// ============================================
// DB_RecipeProgram9 - Checksum Test
// Lines: 254
// CHUNKS: 10 x 100
// Generated by SpinningCam  [2026-08-14 11:34:49]
// ============================================
//
// --- MAKINE AYARLARI ---
// Machine Origin  : X=0.0, Z=0.0
// Axis Direction  : X=NORMAL, Z=NORMAL
// Output Mode     : RADIUS
// G54 Offset      : X=0.0, Z=0.0
// Home            : X=300.0, Z=150.0
// Retract         : X=50.0, Z=50.0
//
// --- PARCA / BLANK ---
// Blank Radius    : 0.0 mm
// Blank Z Shift   : 0.0 mm
// Final Thickness : 2.0 mm
// Min Safety Gap  : 0.0 mm
//
// --- MANDREL POZISYON ---
// Mandrel Offset  : X=0.0, Z=0.0
// Mandrel Rot     : Rx=0.0, Ry=0.0, Rz=0.0
// ============================================

DATA_BLOCK "DB_RecipeProgram9"
{ S7_Optimized_Access := 'FALSE' }
VERSION : 0.2
UNLINKED
NON_RETAIN
    VAR
        Header : "RecipeHeader";
        Lines1  : Array[0..99] of "RecipeLine";  // global lines 0..99
        Lines2  : Array[0..99] of "RecipeLine";  // global lines 100..199
        Lines3  : Array[0..99] of "RecipeLine";  // global lines 200..299
        Lines4  : Array[0..99] of "RecipeLine";  // global lines 300..399
        Lines5  : Array[0..99] of "RecipeLine";  // global lines 400..499
        Lines6  : Array[0..99] of "RecipeLine";  // global lines 500..599
        Lines7  : Array[0..99] of "RecipeLine";  // global lines 600..699
        Lines8  : Array[0..99] of "RecipeLine";  // global lines 700..799
        Lines9  : Array[0..99] of "RecipeLine";  // global lines 800..899
        Lines10 : Array[0..99] of "RecipeLine";  // global lines 900..999
    END_VAR
BEGIN
    // Header
    Header.sName := 'Checksum Test';
    Header.LineCount := 254;
    Header.Valid := TRUE;
    Header.PreScanned := FALSE;
    Header.MinX := 10.000;
    Header.MaxX := 134.500;
    Header.MinZ := 10.200;
    Header.MaxZ := 60.000;

    // --- Tool table (CAM-authored) ---
    Header.ProvidesToolConfig := TRUE;
    Header.ToolCount := 1;
    Header.AutoCalcAngles := TRUE;
    Header.ToolCode_List[1] := 101;
    Header.ToolCode_List[2] := 0;  // unused
    Header.ToolCode_List[3] := 0;  // unused
    Header.ToolCode_List[4] := 0;  // unused
    Header.ToolAngle_List[1] := 0.0;
    Header.ToolAngle_List[2] := 0.0;
    Header.ToolAngle_List[3] := 0.0;
    Header.ToolAngle_List[4] := 0.0;

    // --- Integrity ---
    // Order-sensitive sum over CMD+Param+F of lines 0..LineCount-1.
    // The PLC recomputes it after reassembling the chunks and refuses
    // to run on a mismatch (16#0316). X/Z are excluded on purpose:
    // float32-vs-float64 rounding would eventually cry wolf.
    Header.ProvidesChecksum := TRUE;
    Header.Checksum := 9593624;

    // Recipe Lines (254 total)

    // --- Lines1 (global lines 0..99) ---
    Lines1[0].X := 0.000; Lines1[0].Z := 0.000; Lines1[0].F := 0; Lines1[0].CMD := 20; Lines1[0].Param := 100; // Spindle ON 1000 RPM
    Lines1[1].X := 0.000; Lines1[1].Z := 0.000; Lines1[1].F := 0; Lines1[1].CMD := 10; Lines1[1].Param := 101; // Tool Change T101
    Lines1[2].X := 10.000; Lines1[2].Z := 60.000; Lines1[2].F := 300; Lines1[2].CMD := 1; Lines1[2].Param := 0; // G1 Linear
    Lines1[3].X := 10.500; Lines1[3].Z := 59.800; Lines1[3].F := 300; Lines1[3].CMD := 1; Lines1[3].Param := 0; // G1 Linear
    Lines1[4].X := 11.000; Lines1[4].Z := 59.600; Lines1[4].F := 300; Lines1[4].CMD := 1; Lines1[4].Param := 0; // G1 Linear
    Lines1[5].X := 11.500; Lines1[5].Z := 59.400; Lines1[5].F := 300; Lines1[5].CMD := 1; Lines1[5].Param := 0; // G1 Linear
    Lines1[6].X := 12.000; Lines1[6].Z := 59.200; Lines1[6].F := 300; Lines1[6].CMD := 1; Lines1[6].Param := 0; // G1 Linear
    Lines1[7].X := 12.500; Lines1[7].Z := 59.000; Lines1[7].F := 300; Lines1[7].CMD := 1; Lines1[7].Param := 0; // G1 Linear
    Lines1[8].X := 13.000; Lines1[8].Z := 58.800; Lines1[8].F := 300; Lines1[8].CMD := 1; Lines1[8].Param := 0; // G1 Linear
    Lines1[9].X := 13.500; Lines1[9].Z := 58.600; Lines1[9].F := 300; Lines1[9].CMD := 1; Lines1[9].Param := 0; // G1 Linear
    Lines1[10].X := 14.000; Lines1[10].Z := 58.400; Lines1[10].F := 300; Lines1[10].CMD := 1; Lines1[10].Param := 0; // G1 Linear
    Lines1[11].X := 14.500; Lines1[11].Z := 58.200; Lines1[11].F := 300; Lines1[11].CMD := 1; Lines1[11].Param := 0; // G1 Linear
    Lines1[12].X := 15.000; Lines1[12].Z := 58.000; Lines1[12].F := 300; Lines1[12].CMD := 1; Lines1[12].Param := 0; // G1 Linear
    Lines1[13].X := 15.500; Lines1[13].Z := 57.800; Lines1[13].F := 300; Lines1[13].CMD := 1; Lines1[13].Param := 0; // G1 Linear
    Lines1[14].X := 16.000; Lines1[14].Z := 57.600; Lines1[14].F := 300; Lines1[14].CMD := 1; Lines1[14].Param := 0; // G1 Linear
    Lines1[15].X := 16.500; Lines1[15].Z := 57.400; Lines1[15].F := 300; Lines1[15].CMD := 1; Lines1[15].Param := 0; // G1 Linear
    Lines1[16].X := 17.000; Lines1[16].Z := 57.200; Lines1[16].F := 300; Lines1[16].CMD := 1; Lines1[16].Param := 0; // G1 Linear
    Lines1[17].X := 17.500; Lines1[17].Z := 57.000; Lines1[17].F := 300; Lines1[17].CMD := 1; Lines1[17].Param := 0; // G1 Linear
    Lines1[18].X := 18.000; Lines1[18].Z := 56.800; Lines1[18].F := 300; Lines1[18].CMD := 1; Lines1[18].Param := 0; // G1 Linear
    Lines1[19].X := 18.500; Lines1[19].Z := 56.600; Lines1[19].F := 300; Lines1[19].CMD := 1; Lines1[19].Param := 0; // G1 Linear
    Lines1[20].X := 19.000; Lines1[20].Z := 56.400; Lines1[20].F := 300; Lines1[20].CMD := 1; Lines1[20].Param := 0; // G1 Linear
    Lines1[21].X := 19.500; Lines1[21].Z := 56.200; Lines1[21].F := 300; Lines1[21].CMD := 1; Lines1[21].Param := 0; // G1 Linear
    Lines1[22].X := 20.000; Lines1[22].Z := 56.000; Lines1[22].F := 300; Lines1[22].CMD := 1; Lines1[22].Param := 0; // G1 Linear
    Lines1[23].X := 20.500; Lines1[23].Z := 55.800; Lines1[23].F := 300; Lines1[23].CMD := 1; Lines1[23].Param := 0; // G1 Linear
    Lines1[24].X := 21.000; Lines1[24].Z := 55.600; Lines1[24].F := 300; Lines1[24].CMD := 1; Lines1[24].Param := 0; // G1 Linear
    Lines1[25].X := 21.500; Lines1[25].Z := 55.400; Lines1[25].F := 300; Lines1[25].CMD := 1; Lines1[25].Param := 0; // G1 Linear
    Lines1[26].X := 22.000; Lines1[26].Z := 55.200; Lines1[26].F := 300; Lines1[26].CMD := 1; Lines1[26].Param := 0; // G1 Linear
    Lines1[27].X := 22.500; Lines1[27].Z := 55.000; Lines1[27].F := 300; Lines1[27].CMD := 1; Lines1[27].Param := 0; // G1 Linear
    Lines1[28].X := 23.000; Lines1[28].Z := 54.800; Lines1[28].F := 300; Lines1[28].CMD := 1; Lines1[28].Param := 0; // G1 Linear
    Lines1[29].X := 23.500; Lines1[29].Z := 54.600; Lines1[29].F := 300; Lines1[29].CMD := 1; Lines1[29].Param := 0; // G1 Linear
    Lines1[30].X := 24.000; Lines1[30].Z := 54.400; Lines1[30].F := 300; Lines1[30].CMD := 1; Lines1[30].Param := 0; // G1 Linear
    Lines1[31].X := 24.500; Lines1[31].Z := 54.200; Lines1[31].F := 300; Lines1[31].CMD := 1; Lines1[31].Param := 0; // G1 Linear
    Lines1[32].X := 25.000; Lines1[32].Z := 54.000; Lines1[32].F := 300; Lines1[32].CMD := 1; Lines1[32].Param := 0; // G1 Linear
    Lines1[33].X := 25.500; Lines1[33].Z := 53.800; Lines1[33].F := 300; Lines1[33].CMD := 1; Lines1[33].Param := 0; // G1 Linear
    Lines1[34].X := 26.000; Lines1[34].Z := 53.600; Lines1[34].F := 300; Lines1[34].CMD := 1; Lines1[34].Param := 0; // G1 Linear
    Lines1[35].X := 26.500; Lines1[35].Z := 53.400; Lines1[35].F := 300; Lines1[35].CMD := 1; Lines1[35].Param := 0; // G1 Linear
    Lines1[36].X := 27.000; Lines1[36].Z := 53.200; Lines1[36].F := 300; Lines1[36].CMD := 1; Lines1[36].Param := 0; // G1 Linear
    Lines1[37].X := 27.500; Lines1[37].Z := 53.000; Lines1[37].F := 300; Lines1[37].CMD := 1; Lines1[37].Param := 0; // G1 Linear
    Lines1[38].X := 28.000; Lines1[38].Z := 52.800; Lines1[38].F := 300; Lines1[38].CMD := 1; Lines1[38].Param := 0; // G1 Linear
    Lines1[39].X := 28.500; Lines1[39].Z := 52.600; Lines1[39].F := 300; Lines1[39].CMD := 1; Lines1[39].Param := 0; // G1 Linear
    Lines1[40].X := 29.000; Lines1[40].Z := 52.400; Lines1[40].F := 300; Lines1[40].CMD := 1; Lines1[40].Param := 0; // G1 Linear
    Lines1[41].X := 29.500; Lines1[41].Z := 52.200; Lines1[41].F := 300; Lines1[41].CMD := 1; Lines1[41].Param := 0; // G1 Linear
    Lines1[42].X := 30.000; Lines1[42].Z := 52.000; Lines1[42].F := 300; Lines1[42].CMD := 1; Lines1[42].Param := 0; // G1 Linear
    Lines1[43].X := 30.500; Lines1[43].Z := 51.800; Lines1[43].F := 300; Lines1[43].CMD := 1; Lines1[43].Param := 0; // G1 Linear
    Lines1[44].X := 31.000; Lines1[44].Z := 51.600; Lines1[44].F := 300; Lines1[44].CMD := 1; Lines1[44].Param := 0; // G1 Linear
    Lines1[45].X := 31.500; Lines1[45].Z := 51.400; Lines1[45].F := 300; Lines1[45].CMD := 1; Lines1[45].Param := 0; // G1 Linear
    Lines1[46].X := 32.000; Lines1[46].Z := 51.200; Lines1[46].F := 300; Lines1[46].CMD := 1; Lines1[46].Param := 0; // G1 Linear
    Lines1[47].X := 32.500; Lines1[47].Z := 51.000; Lines1[47].F := 300; Lines1[47].CMD := 1; Lines1[47].Param := 0; // G1 Linear
    Lines1[48].X := 33.000; Lines1[48].Z := 50.800; Lines1[48].F := 300; Lines1[48].CMD := 1; Lines1[48].Param := 0; // G1 Linear
    Lines1[49].X := 33.500; Lines1[49].Z := 50.600; Lines1[49].F := 300; Lines1[49].CMD := 1; Lines1[49].Param := 0; // G1 Linear
    Lines1[50].X := 34.000; Lines1[50].Z := 50.400; Lines1[50].F := 300; Lines1[50].CMD := 1; Lines1[50].Param := 0; // G1 Linear
    Lines1[51].X := 34.500; Lines1[51].Z := 50.200; Lines1[51].F := 300; Lines1[51].CMD := 1; Lines1[51].Param := 0; // G1 Linear
    Lines1[52].X := 35.000; Lines1[52].Z := 50.000; Lines1[52].F := 300; Lines1[52].CMD := 1; Lines1[52].Param := 0; // G1 Linear
    Lines1[53].X := 35.500; Lines1[53].Z := 49.800; Lines1[53].F := 300; Lines1[53].CMD := 1; Lines1[53].Param := 0; // G1 Linear
    Lines1[54].X := 36.000; Lines1[54].Z := 49.600; Lines1[54].F := 300; Lines1[54].CMD := 1; Lines1[54].Param := 0; // G1 Linear
    Lines1[55].X := 36.500; Lines1[55].Z := 49.400; Lines1[55].F := 300; Lines1[55].CMD := 1; Lines1[55].Param := 0; // G1 Linear
    Lines1[56].X := 37.000; Lines1[56].Z := 49.200; Lines1[56].F := 300; Lines1[56].CMD := 1; Lines1[56].Param := 0; // G1 Linear
    Lines1[57].X := 37.500; Lines1[57].Z := 49.000; Lines1[57].F := 300; Lines1[57].CMD := 1; Lines1[57].Param := 0; // G1 Linear
    Lines1[58].X := 38.000; Lines1[58].Z := 48.800; Lines1[58].F := 300; Lines1[58].CMD := 1; Lines1[58].Param := 0; // G1 Linear
    Lines1[59].X := 38.500; Lines1[59].Z := 48.600; Lines1[59].F := 300; Lines1[59].CMD := 1; Lines1[59].Param := 0; // G1 Linear
    Lines1[60].X := 39.000; Lines1[60].Z := 48.400; Lines1[60].F := 300; Lines1[60].CMD := 1; Lines1[60].Param := 0; // G1 Linear
    Lines1[61].X := 39.500; Lines1[61].Z := 48.200; Lines1[61].F := 300; Lines1[61].CMD := 1; Lines1[61].Param := 0; // G1 Linear
    Lines1[62].X := 40.000; Lines1[62].Z := 48.000; Lines1[62].F := 300; Lines1[62].CMD := 1; Lines1[62].Param := 0; // G1 Linear
    Lines1[63].X := 40.500; Lines1[63].Z := 47.800; Lines1[63].F := 300; Lines1[63].CMD := 1; Lines1[63].Param := 0; // G1 Linear
    Lines1[64].X := 41.000; Lines1[64].Z := 47.600; Lines1[64].F := 300; Lines1[64].CMD := 1; Lines1[64].Param := 0; // G1 Linear
    Lines1[65].X := 41.500; Lines1[65].Z := 47.400; Lines1[65].F := 300; Lines1[65].CMD := 1; Lines1[65].Param := 0; // G1 Linear
    Lines1[66].X := 42.000; Lines1[66].Z := 47.200; Lines1[66].F := 300; Lines1[66].CMD := 1; Lines1[66].Param := 0; // G1 Linear
    Lines1[67].X := 42.500; Lines1[67].Z := 47.000; Lines1[67].F := 300; Lines1[67].CMD := 1; Lines1[67].Param := 0; // G1 Linear
    Lines1[68].X := 43.000; Lines1[68].Z := 46.800; Lines1[68].F := 300; Lines1[68].CMD := 1; Lines1[68].Param := 0; // G1 Linear
    Lines1[69].X := 43.500; Lines1[69].Z := 46.600; Lines1[69].F := 300; Lines1[69].CMD := 1; Lines1[69].Param := 0; // G1 Linear
    Lines1[70].X := 44.000; Lines1[70].Z := 46.400; Lines1[70].F := 300; Lines1[70].CMD := 1; Lines1[70].Param := 0; // G1 Linear
    Lines1[71].X := 44.500; Lines1[71].Z := 46.200; Lines1[71].F := 300; Lines1[71].CMD := 1; Lines1[71].Param := 0; // G1 Linear
    Lines1[72].X := 45.000; Lines1[72].Z := 46.000; Lines1[72].F := 300; Lines1[72].CMD := 1; Lines1[72].Param := 0; // G1 Linear
    Lines1[73].X := 45.500; Lines1[73].Z := 45.800; Lines1[73].F := 300; Lines1[73].CMD := 1; Lines1[73].Param := 0; // G1 Linear
    Lines1[74].X := 46.000; Lines1[74].Z := 45.600; Lines1[74].F := 300; Lines1[74].CMD := 1; Lines1[74].Param := 0; // G1 Linear
    Lines1[75].X := 46.500; Lines1[75].Z := 45.400; Lines1[75].F := 300; Lines1[75].CMD := 1; Lines1[75].Param := 0; // G1 Linear
    Lines1[76].X := 47.000; Lines1[76].Z := 45.200; Lines1[76].F := 300; Lines1[76].CMD := 1; Lines1[76].Param := 0; // G1 Linear
    Lines1[77].X := 47.500; Lines1[77].Z := 45.000; Lines1[77].F := 300; Lines1[77].CMD := 1; Lines1[77].Param := 0; // G1 Linear
    Lines1[78].X := 48.000; Lines1[78].Z := 44.800; Lines1[78].F := 300; Lines1[78].CMD := 1; Lines1[78].Param := 0; // G1 Linear
    Lines1[79].X := 48.500; Lines1[79].Z := 44.600; Lines1[79].F := 300; Lines1[79].CMD := 1; Lines1[79].Param := 0; // G1 Linear
    Lines1[80].X := 49.000; Lines1[80].Z := 44.400; Lines1[80].F := 300; Lines1[80].CMD := 1; Lines1[80].Param := 0; // G1 Linear
    Lines1[81].X := 49.500; Lines1[81].Z := 44.200; Lines1[81].F := 300; Lines1[81].CMD := 1; Lines1[81].Param := 0; // G1 Linear
    Lines1[82].X := 50.000; Lines1[82].Z := 44.000; Lines1[82].F := 300; Lines1[82].CMD := 1; Lines1[82].Param := 0; // G1 Linear
    Lines1[83].X := 50.500; Lines1[83].Z := 43.800; Lines1[83].F := 300; Lines1[83].CMD := 1; Lines1[83].Param := 0; // G1 Linear
    Lines1[84].X := 51.000; Lines1[84].Z := 43.600; Lines1[84].F := 300; Lines1[84].CMD := 1; Lines1[84].Param := 0; // G1 Linear
    Lines1[85].X := 51.500; Lines1[85].Z := 43.400; Lines1[85].F := 300; Lines1[85].CMD := 1; Lines1[85].Param := 0; // G1 Linear
    Lines1[86].X := 52.000; Lines1[86].Z := 43.200; Lines1[86].F := 300; Lines1[86].CMD := 1; Lines1[86].Param := 0; // G1 Linear
    Lines1[87].X := 52.500; Lines1[87].Z := 43.000; Lines1[87].F := 300; Lines1[87].CMD := 1; Lines1[87].Param := 0; // G1 Linear
    Lines1[88].X := 53.000; Lines1[88].Z := 42.800; Lines1[88].F := 300; Lines1[88].CMD := 1; Lines1[88].Param := 0; // G1 Linear
    Lines1[89].X := 53.500; Lines1[89].Z := 42.600; Lines1[89].F := 300; Lines1[89].CMD := 1; Lines1[89].Param := 0; // G1 Linear
    Lines1[90].X := 54.000; Lines1[90].Z := 42.400; Lines1[90].F := 300; Lines1[90].CMD := 1; Lines1[90].Param := 0; // G1 Linear
    Lines1[91].X := 54.500; Lines1[91].Z := 42.200; Lines1[91].F := 300; Lines1[91].CMD := 1; Lines1[91].Param := 0; // G1 Linear
    Lines1[92].X := 55.000; Lines1[92].Z := 42.000; Lines1[92].F := 300; Lines1[92].CMD := 1; Lines1[92].Param := 0; // G1 Linear
    Lines1[93].X := 55.500; Lines1[93].Z := 41.800; Lines1[93].F := 300; Lines1[93].CMD := 1; Lines1[93].Param := 0; // G1 Linear
    Lines1[94].X := 56.000; Lines1[94].Z := 41.600; Lines1[94].F := 300; Lines1[94].CMD := 1; Lines1[94].Param := 0; // G1 Linear
    Lines1[95].X := 56.500; Lines1[95].Z := 41.400; Lines1[95].F := 300; Lines1[95].CMD := 1; Lines1[95].Param := 0; // G1 Linear
    Lines1[96].X := 57.000; Lines1[96].Z := 41.200; Lines1[96].F := 300; Lines1[96].CMD := 1; Lines1[96].Param := 0; // G1 Linear
    Lines1[97].X := 57.500; Lines1[97].Z := 41.000; Lines1[97].F := 300; Lines1[97].CMD := 1; Lines1[97].Param := 0; // G1 Linear
    Lines1[98].X := 58.000; Lines1[98].Z := 40.800; Lines1[98].F := 300; Lines1[98].CMD := 1; Lines1[98].Param := 0; // G1 Linear
    Lines1[99].X := 58.500; Lines1[99].Z := 40.600; Lines1[99].F := 300; Lines1[99].CMD := 1; Lines1[99].Param := 0; // G1 Linear

    // --- Lines2 (global lines 100..199) ---
    Lines2[0].X := 59.000; Lines2[0].Z := 40.400; Lines2[0].F := 300; Lines2[0].CMD := 1; Lines2[0].Param := 0; // G1 Linear
    Lines2[1].X := 59.500; Lines2[1].Z := 40.200; Lines2[1].F := 300; Lines2[1].CMD := 1; Lines2[1].Param := 0; // G1 Linear
    Lines2[2].X := 60.000; Lines2[2].Z := 40.000; Lines2[2].F := 300; Lines2[2].CMD := 1; Lines2[2].Param := 0; // G1 Linear
    Lines2[3].X := 60.500; Lines2[3].Z := 39.800; Lines2[3].F := 300; Lines2[3].CMD := 1; Lines2[3].Param := 0; // G1 Linear
    Lines2[4].X := 61.000; Lines2[4].Z := 39.600; Lines2[4].F := 300; Lines2[4].CMD := 1; Lines2[4].Param := 0; // G1 Linear
    Lines2[5].X := 61.500; Lines2[5].Z := 39.400; Lines2[5].F := 300; Lines2[5].CMD := 1; Lines2[5].Param := 0; // G1 Linear
    Lines2[6].X := 62.000; Lines2[6].Z := 39.200; Lines2[6].F := 300; Lines2[6].CMD := 1; Lines2[6].Param := 0; // G1 Linear
    Lines2[7].X := 62.500; Lines2[7].Z := 39.000; Lines2[7].F := 300; Lines2[7].CMD := 1; Lines2[7].Param := 0; // G1 Linear
    Lines2[8].X := 63.000; Lines2[8].Z := 38.800; Lines2[8].F := 300; Lines2[8].CMD := 1; Lines2[8].Param := 0; // G1 Linear
    Lines2[9].X := 63.500; Lines2[9].Z := 38.600; Lines2[9].F := 300; Lines2[9].CMD := 1; Lines2[9].Param := 0; // G1 Linear
    Lines2[10].X := 64.000; Lines2[10].Z := 38.400; Lines2[10].F := 300; Lines2[10].CMD := 1; Lines2[10].Param := 0; // G1 Linear
    Lines2[11].X := 64.500; Lines2[11].Z := 38.200; Lines2[11].F := 300; Lines2[11].CMD := 1; Lines2[11].Param := 0; // G1 Linear
    Lines2[12].X := 65.000; Lines2[12].Z := 38.000; Lines2[12].F := 300; Lines2[12].CMD := 1; Lines2[12].Param := 0; // G1 Linear
    Lines2[13].X := 65.500; Lines2[13].Z := 37.800; Lines2[13].F := 300; Lines2[13].CMD := 1; Lines2[13].Param := 0; // G1 Linear
    Lines2[14].X := 66.000; Lines2[14].Z := 37.600; Lines2[14].F := 300; Lines2[14].CMD := 1; Lines2[14].Param := 0; // G1 Linear
    Lines2[15].X := 66.500; Lines2[15].Z := 37.400; Lines2[15].F := 300; Lines2[15].CMD := 1; Lines2[15].Param := 0; // G1 Linear
    Lines2[16].X := 67.000; Lines2[16].Z := 37.200; Lines2[16].F := 300; Lines2[16].CMD := 1; Lines2[16].Param := 0; // G1 Linear
    Lines2[17].X := 67.500; Lines2[17].Z := 37.000; Lines2[17].F := 300; Lines2[17].CMD := 1; Lines2[17].Param := 0; // G1 Linear
    Lines2[18].X := 68.000; Lines2[18].Z := 36.800; Lines2[18].F := 300; Lines2[18].CMD := 1; Lines2[18].Param := 0; // G1 Linear
    Lines2[19].X := 68.500; Lines2[19].Z := 36.600; Lines2[19].F := 300; Lines2[19].CMD := 1; Lines2[19].Param := 0; // G1 Linear
    Lines2[20].X := 69.000; Lines2[20].Z := 36.400; Lines2[20].F := 300; Lines2[20].CMD := 1; Lines2[20].Param := 0; // G1 Linear
    Lines2[21].X := 69.500; Lines2[21].Z := 36.200; Lines2[21].F := 300; Lines2[21].CMD := 1; Lines2[21].Param := 0; // G1 Linear
    Lines2[22].X := 70.000; Lines2[22].Z := 36.000; Lines2[22].F := 300; Lines2[22].CMD := 1; Lines2[22].Param := 0; // G1 Linear
    Lines2[23].X := 70.500; Lines2[23].Z := 35.800; Lines2[23].F := 300; Lines2[23].CMD := 1; Lines2[23].Param := 0; // G1 Linear
    Lines2[24].X := 71.000; Lines2[24].Z := 35.600; Lines2[24].F := 300; Lines2[24].CMD := 1; Lines2[24].Param := 0; // G1 Linear
    Lines2[25].X := 71.500; Lines2[25].Z := 35.400; Lines2[25].F := 300; Lines2[25].CMD := 1; Lines2[25].Param := 0; // G1 Linear
    Lines2[26].X := 72.000; Lines2[26].Z := 35.200; Lines2[26].F := 300; Lines2[26].CMD := 1; Lines2[26].Param := 0; // G1 Linear
    Lines2[27].X := 72.500; Lines2[27].Z := 35.000; Lines2[27].F := 300; Lines2[27].CMD := 1; Lines2[27].Param := 0; // G1 Linear
    Lines2[28].X := 73.000; Lines2[28].Z := 34.800; Lines2[28].F := 300; Lines2[28].CMD := 1; Lines2[28].Param := 0; // G1 Linear
    Lines2[29].X := 73.500; Lines2[29].Z := 34.600; Lines2[29].F := 300; Lines2[29].CMD := 1; Lines2[29].Param := 0; // G1 Linear
    Lines2[30].X := 74.000; Lines2[30].Z := 34.400; Lines2[30].F := 300; Lines2[30].CMD := 1; Lines2[30].Param := 0; // G1 Linear
    Lines2[31].X := 74.500; Lines2[31].Z := 34.200; Lines2[31].F := 300; Lines2[31].CMD := 1; Lines2[31].Param := 0; // G1 Linear
    Lines2[32].X := 75.000; Lines2[32].Z := 34.000; Lines2[32].F := 300; Lines2[32].CMD := 1; Lines2[32].Param := 0; // G1 Linear
    Lines2[33].X := 75.500; Lines2[33].Z := 33.800; Lines2[33].F := 300; Lines2[33].CMD := 1; Lines2[33].Param := 0; // G1 Linear
    Lines2[34].X := 76.000; Lines2[34].Z := 33.600; Lines2[34].F := 300; Lines2[34].CMD := 1; Lines2[34].Param := 0; // G1 Linear
    Lines2[35].X := 76.500; Lines2[35].Z := 33.400; Lines2[35].F := 300; Lines2[35].CMD := 1; Lines2[35].Param := 0; // G1 Linear
    Lines2[36].X := 77.000; Lines2[36].Z := 33.200; Lines2[36].F := 300; Lines2[36].CMD := 1; Lines2[36].Param := 0; // G1 Linear
    Lines2[37].X := 77.500; Lines2[37].Z := 33.000; Lines2[37].F := 300; Lines2[37].CMD := 1; Lines2[37].Param := 0; // G1 Linear
    Lines2[38].X := 78.000; Lines2[38].Z := 32.800; Lines2[38].F := 300; Lines2[38].CMD := 1; Lines2[38].Param := 0; // G1 Linear
    Lines2[39].X := 78.500; Lines2[39].Z := 32.600; Lines2[39].F := 300; Lines2[39].CMD := 1; Lines2[39].Param := 0; // G1 Linear
    Lines2[40].X := 79.000; Lines2[40].Z := 32.400; Lines2[40].F := 300; Lines2[40].CMD := 1; Lines2[40].Param := 0; // G1 Linear
    Lines2[41].X := 79.500; Lines2[41].Z := 32.200; Lines2[41].F := 300; Lines2[41].CMD := 1; Lines2[41].Param := 0; // G1 Linear
    Lines2[42].X := 80.000; Lines2[42].Z := 32.000; Lines2[42].F := 300; Lines2[42].CMD := 1; Lines2[42].Param := 0; // G1 Linear
    Lines2[43].X := 80.500; Lines2[43].Z := 31.800; Lines2[43].F := 300; Lines2[43].CMD := 1; Lines2[43].Param := 0; // G1 Linear
    Lines2[44].X := 81.000; Lines2[44].Z := 31.600; Lines2[44].F := 300; Lines2[44].CMD := 1; Lines2[44].Param := 0; // G1 Linear
    Lines2[45].X := 81.500; Lines2[45].Z := 31.400; Lines2[45].F := 300; Lines2[45].CMD := 1; Lines2[45].Param := 0; // G1 Linear
    Lines2[46].X := 82.000; Lines2[46].Z := 31.200; Lines2[46].F := 300; Lines2[46].CMD := 1; Lines2[46].Param := 0; // G1 Linear
    Lines2[47].X := 82.500; Lines2[47].Z := 31.000; Lines2[47].F := 300; Lines2[47].CMD := 1; Lines2[47].Param := 0; // G1 Linear
    Lines2[48].X := 83.000; Lines2[48].Z := 30.800; Lines2[48].F := 300; Lines2[48].CMD := 1; Lines2[48].Param := 0; // G1 Linear
    Lines2[49].X := 83.500; Lines2[49].Z := 30.600; Lines2[49].F := 300; Lines2[49].CMD := 1; Lines2[49].Param := 0; // G1 Linear
    Lines2[50].X := 84.000; Lines2[50].Z := 30.400; Lines2[50].F := 300; Lines2[50].CMD := 1; Lines2[50].Param := 0; // G1 Linear
    Lines2[51].X := 84.500; Lines2[51].Z := 30.200; Lines2[51].F := 300; Lines2[51].CMD := 1; Lines2[51].Param := 0; // G1 Linear
    Lines2[52].X := 85.000; Lines2[52].Z := 30.000; Lines2[52].F := 300; Lines2[52].CMD := 1; Lines2[52].Param := 0; // G1 Linear
    Lines2[53].X := 85.500; Lines2[53].Z := 29.800; Lines2[53].F := 300; Lines2[53].CMD := 1; Lines2[53].Param := 0; // G1 Linear
    Lines2[54].X := 86.000; Lines2[54].Z := 29.600; Lines2[54].F := 300; Lines2[54].CMD := 1; Lines2[54].Param := 0; // G1 Linear
    Lines2[55].X := 86.500; Lines2[55].Z := 29.400; Lines2[55].F := 300; Lines2[55].CMD := 1; Lines2[55].Param := 0; // G1 Linear
    Lines2[56].X := 87.000; Lines2[56].Z := 29.200; Lines2[56].F := 300; Lines2[56].CMD := 1; Lines2[56].Param := 0; // G1 Linear
    Lines2[57].X := 87.500; Lines2[57].Z := 29.000; Lines2[57].F := 300; Lines2[57].CMD := 1; Lines2[57].Param := 0; // G1 Linear
    Lines2[58].X := 88.000; Lines2[58].Z := 28.800; Lines2[58].F := 300; Lines2[58].CMD := 1; Lines2[58].Param := 0; // G1 Linear
    Lines2[59].X := 88.500; Lines2[59].Z := 28.600; Lines2[59].F := 300; Lines2[59].CMD := 1; Lines2[59].Param := 0; // G1 Linear
    Lines2[60].X := 89.000; Lines2[60].Z := 28.400; Lines2[60].F := 300; Lines2[60].CMD := 1; Lines2[60].Param := 0; // G1 Linear
    Lines2[61].X := 89.500; Lines2[61].Z := 28.200; Lines2[61].F := 300; Lines2[61].CMD := 1; Lines2[61].Param := 0; // G1 Linear
    Lines2[62].X := 90.000; Lines2[62].Z := 28.000; Lines2[62].F := 300; Lines2[62].CMD := 1; Lines2[62].Param := 0; // G1 Linear
    Lines2[63].X := 90.500; Lines2[63].Z := 27.800; Lines2[63].F := 300; Lines2[63].CMD := 1; Lines2[63].Param := 0; // G1 Linear
    Lines2[64].X := 91.000; Lines2[64].Z := 27.600; Lines2[64].F := 300; Lines2[64].CMD := 1; Lines2[64].Param := 0; // G1 Linear
    Lines2[65].X := 91.500; Lines2[65].Z := 27.400; Lines2[65].F := 300; Lines2[65].CMD := 1; Lines2[65].Param := 0; // G1 Linear
    Lines2[66].X := 92.000; Lines2[66].Z := 27.200; Lines2[66].F := 300; Lines2[66].CMD := 1; Lines2[66].Param := 0; // G1 Linear
    Lines2[67].X := 92.500; Lines2[67].Z := 27.000; Lines2[67].F := 300; Lines2[67].CMD := 1; Lines2[67].Param := 0; // G1 Linear
    Lines2[68].X := 93.000; Lines2[68].Z := 26.800; Lines2[68].F := 300; Lines2[68].CMD := 1; Lines2[68].Param := 0; // G1 Linear
    Lines2[69].X := 93.500; Lines2[69].Z := 26.600; Lines2[69].F := 300; Lines2[69].CMD := 1; Lines2[69].Param := 0; // G1 Linear
    Lines2[70].X := 94.000; Lines2[70].Z := 26.400; Lines2[70].F := 300; Lines2[70].CMD := 1; Lines2[70].Param := 0; // G1 Linear
    Lines2[71].X := 94.500; Lines2[71].Z := 26.200; Lines2[71].F := 300; Lines2[71].CMD := 1; Lines2[71].Param := 0; // G1 Linear
    Lines2[72].X := 95.000; Lines2[72].Z := 26.000; Lines2[72].F := 300; Lines2[72].CMD := 1; Lines2[72].Param := 0; // G1 Linear
    Lines2[73].X := 95.500; Lines2[73].Z := 25.800; Lines2[73].F := 300; Lines2[73].CMD := 1; Lines2[73].Param := 0; // G1 Linear
    Lines2[74].X := 96.000; Lines2[74].Z := 25.600; Lines2[74].F := 300; Lines2[74].CMD := 1; Lines2[74].Param := 0; // G1 Linear
    Lines2[75].X := 96.500; Lines2[75].Z := 25.400; Lines2[75].F := 300; Lines2[75].CMD := 1; Lines2[75].Param := 0; // G1 Linear
    Lines2[76].X := 97.000; Lines2[76].Z := 25.200; Lines2[76].F := 300; Lines2[76].CMD := 1; Lines2[76].Param := 0; // G1 Linear
    Lines2[77].X := 97.500; Lines2[77].Z := 25.000; Lines2[77].F := 300; Lines2[77].CMD := 1; Lines2[77].Param := 0; // G1 Linear
    Lines2[78].X := 98.000; Lines2[78].Z := 24.800; Lines2[78].F := 300; Lines2[78].CMD := 1; Lines2[78].Param := 0; // G1 Linear
    Lines2[79].X := 98.500; Lines2[79].Z := 24.600; Lines2[79].F := 300; Lines2[79].CMD := 1; Lines2[79].Param := 0; // G1 Linear
    Lines2[80].X := 99.000; Lines2[80].Z := 24.400; Lines2[80].F := 300; Lines2[80].CMD := 1; Lines2[80].Param := 0; // G1 Linear
    Lines2[81].X := 99.500; Lines2[81].Z := 24.200; Lines2[81].F := 300; Lines2[81].CMD := 1; Lines2[81].Param := 0; // G1 Linear
    Lines2[82].X := 100.000; Lines2[82].Z := 24.000; Lines2[82].F := 300; Lines2[82].CMD := 1; Lines2[82].Param := 0; // G1 Linear
    Lines2[83].X := 100.500; Lines2[83].Z := 23.800; Lines2[83].F := 300; Lines2[83].CMD := 1; Lines2[83].Param := 0; // G1 Linear
    Lines2[84].X := 101.000; Lines2[84].Z := 23.600; Lines2[84].F := 300; Lines2[84].CMD := 1; Lines2[84].Param := 0; // G1 Linear
    Lines2[85].X := 101.500; Lines2[85].Z := 23.400; Lines2[85].F := 300; Lines2[85].CMD := 1; Lines2[85].Param := 0; // G1 Linear
    Lines2[86].X := 102.000; Lines2[86].Z := 23.200; Lines2[86].F := 300; Lines2[86].CMD := 1; Lines2[86].Param := 0; // G1 Linear
    Lines2[87].X := 102.500; Lines2[87].Z := 23.000; Lines2[87].F := 300; Lines2[87].CMD := 1; Lines2[87].Param := 0; // G1 Linear
    Lines2[88].X := 103.000; Lines2[88].Z := 22.800; Lines2[88].F := 300; Lines2[88].CMD := 1; Lines2[88].Param := 0; // G1 Linear
    Lines2[89].X := 103.500; Lines2[89].Z := 22.600; Lines2[89].F := 300; Lines2[89].CMD := 1; Lines2[89].Param := 0; // G1 Linear
    Lines2[90].X := 104.000; Lines2[90].Z := 22.400; Lines2[90].F := 300; Lines2[90].CMD := 1; Lines2[90].Param := 0; // G1 Linear
    Lines2[91].X := 104.500; Lines2[91].Z := 22.200; Lines2[91].F := 300; Lines2[91].CMD := 1; Lines2[91].Param := 0; // G1 Linear
    Lines2[92].X := 105.000; Lines2[92].Z := 22.000; Lines2[92].F := 300; Lines2[92].CMD := 1; Lines2[92].Param := 0; // G1 Linear
    Lines2[93].X := 105.500; Lines2[93].Z := 21.800; Lines2[93].F := 300; Lines2[93].CMD := 1; Lines2[93].Param := 0; // G1 Linear
    Lines2[94].X := 106.000; Lines2[94].Z := 21.600; Lines2[94].F := 300; Lines2[94].CMD := 1; Lines2[94].Param := 0; // G1 Linear
    Lines2[95].X := 106.500; Lines2[95].Z := 21.400; Lines2[95].F := 300; Lines2[95].CMD := 1; Lines2[95].Param := 0; // G1 Linear
    Lines2[96].X := 107.000; Lines2[96].Z := 21.200; Lines2[96].F := 300; Lines2[96].CMD := 1; Lines2[96].Param := 0; // G1 Linear
    Lines2[97].X := 107.500; Lines2[97].Z := 21.000; Lines2[97].F := 300; Lines2[97].CMD := 1; Lines2[97].Param := 0; // G1 Linear
    Lines2[98].X := 108.000; Lines2[98].Z := 20.800; Lines2[98].F := 300; Lines2[98].CMD := 1; Lines2[98].Param := 0; // G1 Linear
    Lines2[99].X := 108.500; Lines2[99].Z := 20.600; Lines2[99].F := 300; Lines2[99].CMD := 1; Lines2[99].Param := 0; // G1 Linear

    // --- Lines3 (global lines 200..253) ---
    Lines3[0].X := 109.000; Lines3[0].Z := 20.400; Lines3[0].F := 300; Lines3[0].CMD := 1; Lines3[0].Param := 0; // G1 Linear
    Lines3[1].X := 109.500; Lines3[1].Z := 20.200; Lines3[1].F := 300; Lines3[1].CMD := 1; Lines3[1].Param := 0; // G1 Linear
    Lines3[2].X := 110.000; Lines3[2].Z := 20.000; Lines3[2].F := 300; Lines3[2].CMD := 1; Lines3[2].Param := 0; // G1 Linear
    Lines3[3].X := 110.500; Lines3[3].Z := 19.800; Lines3[3].F := 300; Lines3[3].CMD := 1; Lines3[3].Param := 0; // G1 Linear
    Lines3[4].X := 111.000; Lines3[4].Z := 19.600; Lines3[4].F := 300; Lines3[4].CMD := 1; Lines3[4].Param := 0; // G1 Linear
    Lines3[5].X := 111.500; Lines3[5].Z := 19.400; Lines3[5].F := 300; Lines3[5].CMD := 1; Lines3[5].Param := 0; // G1 Linear
    Lines3[6].X := 112.000; Lines3[6].Z := 19.200; Lines3[6].F := 300; Lines3[6].CMD := 1; Lines3[6].Param := 0; // G1 Linear
    Lines3[7].X := 112.500; Lines3[7].Z := 19.000; Lines3[7].F := 300; Lines3[7].CMD := 1; Lines3[7].Param := 0; // G1 Linear
    Lines3[8].X := 113.000; Lines3[8].Z := 18.800; Lines3[8].F := 300; Lines3[8].CMD := 1; Lines3[8].Param := 0; // G1 Linear
    Lines3[9].X := 113.500; Lines3[9].Z := 18.600; Lines3[9].F := 300; Lines3[9].CMD := 1; Lines3[9].Param := 0; // G1 Linear
    Lines3[10].X := 114.000; Lines3[10].Z := 18.400; Lines3[10].F := 300; Lines3[10].CMD := 1; Lines3[10].Param := 0; // G1 Linear
    Lines3[11].X := 114.500; Lines3[11].Z := 18.200; Lines3[11].F := 300; Lines3[11].CMD := 1; Lines3[11].Param := 0; // G1 Linear
    Lines3[12].X := 115.000; Lines3[12].Z := 18.000; Lines3[12].F := 300; Lines3[12].CMD := 1; Lines3[12].Param := 0; // G1 Linear
    Lines3[13].X := 115.500; Lines3[13].Z := 17.800; Lines3[13].F := 300; Lines3[13].CMD := 1; Lines3[13].Param := 0; // G1 Linear
    Lines3[14].X := 116.000; Lines3[14].Z := 17.600; Lines3[14].F := 300; Lines3[14].CMD := 1; Lines3[14].Param := 0; // G1 Linear
    Lines3[15].X := 116.500; Lines3[15].Z := 17.400; Lines3[15].F := 300; Lines3[15].CMD := 1; Lines3[15].Param := 0; // G1 Linear
    Lines3[16].X := 117.000; Lines3[16].Z := 17.200; Lines3[16].F := 300; Lines3[16].CMD := 1; Lines3[16].Param := 0; // G1 Linear
    Lines3[17].X := 117.500; Lines3[17].Z := 17.000; Lines3[17].F := 300; Lines3[17].CMD := 1; Lines3[17].Param := 0; // G1 Linear
    Lines3[18].X := 118.000; Lines3[18].Z := 16.800; Lines3[18].F := 300; Lines3[18].CMD := 1; Lines3[18].Param := 0; // G1 Linear
    Lines3[19].X := 118.500; Lines3[19].Z := 16.600; Lines3[19].F := 300; Lines3[19].CMD := 1; Lines3[19].Param := 0; // G1 Linear
    Lines3[20].X := 119.000; Lines3[20].Z := 16.400; Lines3[20].F := 300; Lines3[20].CMD := 1; Lines3[20].Param := 0; // G1 Linear
    Lines3[21].X := 119.500; Lines3[21].Z := 16.200; Lines3[21].F := 300; Lines3[21].CMD := 1; Lines3[21].Param := 0; // G1 Linear
    Lines3[22].X := 120.000; Lines3[22].Z := 16.000; Lines3[22].F := 300; Lines3[22].CMD := 1; Lines3[22].Param := 0; // G1 Linear
    Lines3[23].X := 120.500; Lines3[23].Z := 15.800; Lines3[23].F := 300; Lines3[23].CMD := 1; Lines3[23].Param := 0; // G1 Linear
    Lines3[24].X := 121.000; Lines3[24].Z := 15.600; Lines3[24].F := 300; Lines3[24].CMD := 1; Lines3[24].Param := 0; // G1 Linear
    Lines3[25].X := 121.500; Lines3[25].Z := 15.400; Lines3[25].F := 300; Lines3[25].CMD := 1; Lines3[25].Param := 0; // G1 Linear
    Lines3[26].X := 122.000; Lines3[26].Z := 15.200; Lines3[26].F := 300; Lines3[26].CMD := 1; Lines3[26].Param := 0; // G1 Linear
    Lines3[27].X := 122.500; Lines3[27].Z := 15.000; Lines3[27].F := 300; Lines3[27].CMD := 1; Lines3[27].Param := 0; // G1 Linear
    Lines3[28].X := 123.000; Lines3[28].Z := 14.800; Lines3[28].F := 300; Lines3[28].CMD := 1; Lines3[28].Param := 0; // G1 Linear
    Lines3[29].X := 123.500; Lines3[29].Z := 14.600; Lines3[29].F := 300; Lines3[29].CMD := 1; Lines3[29].Param := 0; // G1 Linear
    Lines3[30].X := 124.000; Lines3[30].Z := 14.400; Lines3[30].F := 300; Lines3[30].CMD := 1; Lines3[30].Param := 0; // G1 Linear
    Lines3[31].X := 124.500; Lines3[31].Z := 14.200; Lines3[31].F := 300; Lines3[31].CMD := 1; Lines3[31].Param := 0; // G1 Linear
    Lines3[32].X := 125.000; Lines3[32].Z := 14.000; Lines3[32].F := 300; Lines3[32].CMD := 1; Lines3[32].Param := 0; // G1 Linear
    Lines3[33].X := 125.500; Lines3[33].Z := 13.800; Lines3[33].F := 300; Lines3[33].CMD := 1; Lines3[33].Param := 0; // G1 Linear
    Lines3[34].X := 126.000; Lines3[34].Z := 13.600; Lines3[34].F := 300; Lines3[34].CMD := 1; Lines3[34].Param := 0; // G1 Linear
    Lines3[35].X := 126.500; Lines3[35].Z := 13.400; Lines3[35].F := 300; Lines3[35].CMD := 1; Lines3[35].Param := 0; // G1 Linear
    Lines3[36].X := 127.000; Lines3[36].Z := 13.200; Lines3[36].F := 300; Lines3[36].CMD := 1; Lines3[36].Param := 0; // G1 Linear
    Lines3[37].X := 127.500; Lines3[37].Z := 13.000; Lines3[37].F := 300; Lines3[37].CMD := 1; Lines3[37].Param := 0; // G1 Linear
    Lines3[38].X := 128.000; Lines3[38].Z := 12.800; Lines3[38].F := 300; Lines3[38].CMD := 1; Lines3[38].Param := 0; // G1 Linear
    Lines3[39].X := 128.500; Lines3[39].Z := 12.600; Lines3[39].F := 300; Lines3[39].CMD := 1; Lines3[39].Param := 0; // G1 Linear
    Lines3[40].X := 129.000; Lines3[40].Z := 12.400; Lines3[40].F := 300; Lines3[40].CMD := 1; Lines3[40].Param := 0; // G1 Linear
    Lines3[41].X := 129.500; Lines3[41].Z := 12.200; Lines3[41].F := 300; Lines3[41].CMD := 1; Lines3[41].Param := 0; // G1 Linear
    Lines3[42].X := 130.000; Lines3[42].Z := 12.000; Lines3[42].F := 300; Lines3[42].CMD := 1; Lines3[42].Param := 0; // G1 Linear
    Lines3[43].X := 130.500; Lines3[43].Z := 11.800; Lines3[43].F := 300; Lines3[43].CMD := 1; Lines3[43].Param := 0; // G1 Linear
    Lines3[44].X := 131.000; Lines3[44].Z := 11.600; Lines3[44].F := 300; Lines3[44].CMD := 1; Lines3[44].Param := 0; // G1 Linear
    Lines3[45].X := 131.500; Lines3[45].Z := 11.400; Lines3[45].F := 300; Lines3[45].CMD := 1; Lines3[45].Param := 0; // G1 Linear
    Lines3[46].X := 132.000; Lines3[46].Z := 11.200; Lines3[46].F := 300; Lines3[46].CMD := 1; Lines3[46].Param := 0; // G1 Linear
    Lines3[47].X := 132.500; Lines3[47].Z := 11.000; Lines3[47].F := 300; Lines3[47].CMD := 1; Lines3[47].Param := 0; // G1 Linear
    Lines3[48].X := 133.000; Lines3[48].Z := 10.800; Lines3[48].F := 300; Lines3[48].CMD := 1; Lines3[48].Param := 0; // G1 Linear
    Lines3[49].X := 133.500; Lines3[49].Z := 10.600; Lines3[49].F := 300; Lines3[49].CMD := 1; Lines3[49].Param := 0; // G1 Linear
    Lines3[50].X := 134.000; Lines3[50].Z := 10.400; Lines3[50].F := 300; Lines3[50].CMD := 1; Lines3[50].Param := 0; // G1 Linear
    Lines3[51].X := 134.500; Lines3[51].Z := 10.200; Lines3[51].F := 300; Lines3[51].CMD := 1; Lines3[51].Param := 0; // G1 Linear
    Lines3[52].X := 134.500; Lines3[52].Z := 10.200; Lines3[52].F := 0; Lines3[52].CMD := 21; Lines3[52].Param := 0; // Spindle OFF
    Lines3[53].X := 0.000; Lines3[53].Z := 0.000; Lines3[53].F := 0; Lines3[53].CMD := 99; Lines3[53].Param := 0; // Program END
END_DATA_BLOCK